RoboDK station: InvertedRobot002.rdk

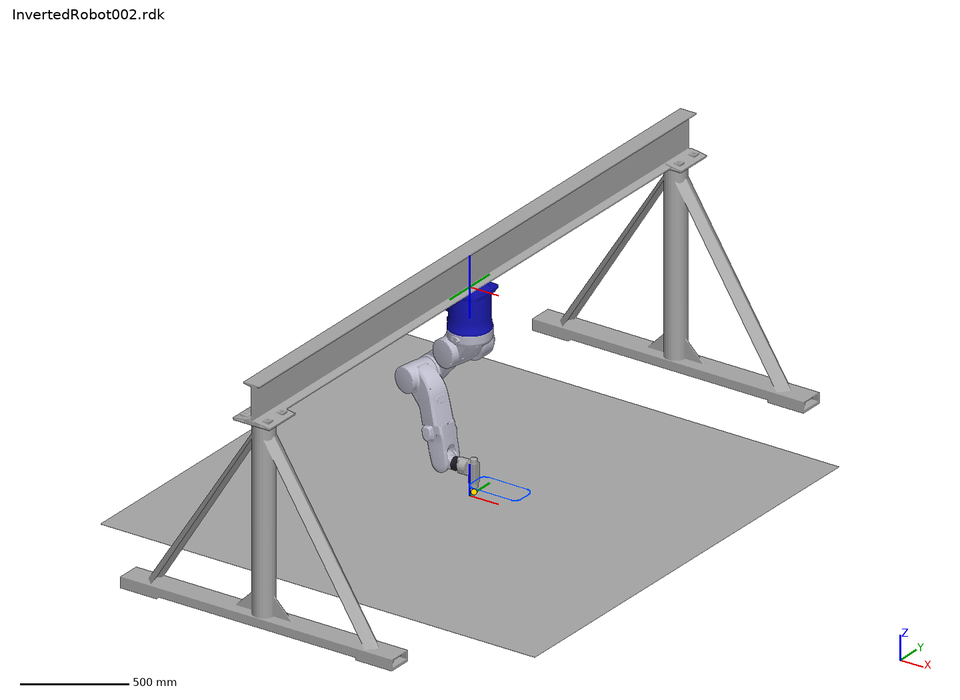
[picture v0: the station drawn from its stored meshes, robots at their saved joint values, targets as dots, program paths as lines]
Station InvertedRobot002 (saved by RoboDK 5.5.4). Poses are relative to the parent item; angles as X-Y-Z fixed-axis rotations.
Station parameters (name, value as stored): TAGS, ['Additive Manufacturing', 'Additive manufacturing'], LIN64
  - frame Denso 1 at (0, 0, 1066.8) mm, rotated rx -180 ry 0 rz 0 deg
    - robot Denso VS-6577G-B: 6 axes, payload 7 kg, reach 854 mm, repeatability 0.03 mm, weight 36 kg
        modified DH rows (alpha deg, a mm, theta deg, d mm): 0, 0, 0, 335; -90, 75, -90, 0; 0, 365, -90, 0; -90, 90, 0, 405; 90, 0, 0, 0; -90, 0, 0, 80
        joint limits [-170, -100, -119, -190, -120, -360] to [170, 135, 169, 190, 120, 360]; home [0, 0, 90, 0, 0, 0]; saved at [-167.935, 49.291, -63.192, 167.582, 76.412, 2.961]
      - tool nozzle, TCP at (110, 0, 80) mm, rotated rx 0 ry 90 rz 0 deg, size 158.8 x 76.2 x 114.9 mm, geometry from nozzle.STEP
      - tool nozzle002, TCP at (100, 0, 80) mm, rotated rx 0 ry 90 rz 0 deg, size 152.4 x 76.2 x 110.1 mm, geometry from nozzle002.STEP
  - frame Ref001 at (0, 0, 0) mm
    - object Part at (0, 0, 0) mm, size 120 x 120 x 160 mm, geometry from part.sld
  - machining project Print3D settings: /home/iRETI/RoboticsResearch/WallSections/12x12x0.875.gcode | rotZ(0) | rotX(0)*rotY(0) | rotZ(0) | on%PROGNAME%_Start | Extruder(-1) | on%PROGNAME%_Approach | on%PROGNAME%_Activate | on%PROGNAME%_Retract | on%PROGNAME%_Finish | SetRPM(%1) | SetTool(%1) | Extruder(%1) | OutOn(%1) | OutOff(%1) | OutOnMov(%1) | OutOffMov(%1) | Extruder(-1) | M_RunCode(%1)
  - program Print3D (292 instructions, listed below)
  - Python program Extruder (listed below)
  - Python program SimulateFinalResult (listed below)
  - frame Frame 4 at (0, 0, 1066.8) mm
    - object GantryAssembly at (0, 0, 0) mm, size 1524 x 3505.2 x 1270 mm, geometry from GantryAssembly.STEP
  - frame Frame 5 at (0, 0, 0) mm
    - object GarageFloor at (0, 0, 0) mm, size 2438.4 x 2438.4 x 2.5 mm, geometry from GarageFloor.STEP
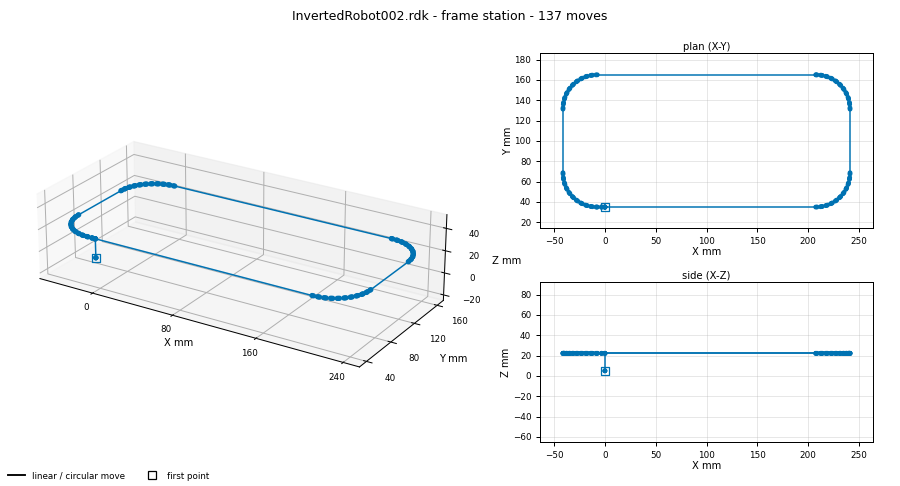
[picture p0: tool path of InvertedRobot002.rdk in frame station, 137 of 137 moves have a stored position in this frame; points joined in program order, loops and branches not executed]

--- program Print3D (robot Denso VS-6577G-B) ---
  Smooth(1)
  Call M_RunCode(107)
  Call M_RunCode(104)
  Set speed (83.3 mm/s)
  Set speed (1000.0 mm/s)
  Set Ref.: Ref001
  Set Tool: nozzle002
  Show nozzle002
  MoveJ 1 to (0, 34.91, 5) mm, rotated rx 180 ry 0 rz 180 deg; joints [-167.691, 46.522, -59.109, 167.397, 77.707, 2.725]
  MoveL 2 to (0, 34.91, 5) mm, rotated rx 180 ry 0 rz 180 deg; joints [-167.691, 46.522, -59.109, 167.397, 77.707, 2.725]
  Call Extruder(-1)
  MoveL 3 to (0, 34.91, 5) mm, rotated rx 180 ry 0 rz 180 deg; joints [-167.691, 46.522, -59.109, 167.397, 77.707, 2.725]
  Call M_RunCode(109)
  Call M_RunCode(82)
  Call Extruder(0.00000)
  Set speed (130.0 mm/s)
  MoveL 4 to (0, 34.91, 22.22) mm, rotated rx -180 ry 0 rz 180 deg; joints [-167.691, 49.055, -63.307, 167.313, 76.082, 3.099]
  Call Extruder(-2.00000)
  Set speed (40.0 mm/s)
  MoveL 5 to (0, 34.91, 22.22) mm, rotated rx -180 ry 0 rz 180 deg; joints [-167.691, 49.055, -63.307, 167.313, 76.082, 3.099]
  Call Extruder(0.00000)
  Set speed (130.0 mm/s)
  MoveL 6 to (0, 34.91, 22.22) mm, rotated rx -180 ry 0 rz 180 deg; joints [-167.691, 49.055, -63.307, 167.313, 76.082, 3.099]
  Call Extruder(2.00000)
  Set speed (40.0 mm/s)
  MoveL 7 to (0, 34.91, 22.22) mm, rotated rx -180 ry 0 rz 180 deg; joints [-167.691, 49.055, -63.307, 167.313, 76.082, 3.099]
  Set speed (30.0 mm/s)
  MoveL 8 to (0, 34.91, 22.22) mm, rotated rx -180 ry 0 rz 180 deg; joints [-167.691, 49.055, -63.307, 167.313, 76.082, 3.099]
  Call Extruder(209.10557)
  MoveL 9 to (207.51, 34.91, 22.23) mm, rotated rx -180 ry 0 rz 180 deg; joints [-36.308, 40.081, -64.789, 38.967, 109.685, 15.241]
  Call Extruder(210.41057)
  MoveL 10 to (208.82, 34.98, 22.22) mm, rotated rx 180 ry 0 rz -180 deg; joints [-35.623, 40.188, -64.796, 38.243, 109.785, 14.937]
  Call Extruder(213.89122)
  MoveL 11 to (212.3, 35.25, 22.22) mm, rotated rx -180 ry 0 rz 180 deg; joints [-33.986, 40.479, -64.812, 36.496, 109.977, 14.186]
  Call Extruder(214.76022)
  MoveL 12 to (213.16, 35.34, 22.22) mm, rotated rx -180 ry 0 rz 180 deg; joints [-33.614, 40.553, -64.815, 36.098, 110.011, 14.01]
  Call Extruder(215.62924)
  MoveL 13 to (214.01, 35.53, 22.22) mm, rotated rx -180 ry 0 rz 180 deg; joints [-33.334, 40.631, -64.819, 35.793, 110.018, 13.864]
  Call Extruder(219.10988)
  MoveL 14 to (217.4, 36.34, 22.22) mm, rotated rx 180 ry 0 rz -180 deg; joints [-32.337, 40.947, -64.83, 34.697, 110.004, 13.325]
  Call Extruder(219.97888)
  MoveL 15 to (218.25, 36.56, 22.23) mm, rotated rx -180 ry 0 rz 180 deg; joints [-32.115, 41.026, -64.832, 34.452, 109.991, 13.2]
  Call Extruder(220.84782)
  MoveL 16 to (219.06, 36.88, 22.23) mm, rotated rx -180 ry 0 rz 180 deg; joints [-31.983, 41.107, -64.834, 34.298, 109.956, 13.105]
  Call Extruder(224.32848)
  MoveL 17 to (222.28, 38.21, 22.22) mm, rotated rx -180 ry 0 rz 180 deg; joints [-31.532, 41.434, -64.839, 33.766, 109.79, 12.755]
  Call Extruder(225.19749)
  MoveL 18 to (223.08, 38.56, 22.22) mm, rotated rx 180 ry 0 rz 180 deg; joints [-31.439, 41.515, -64.839, 33.653, 109.743, 12.674]
  Call Extruder(226.06647)
  MoveL 19 to (223.83, 39, 22.22) mm, rotated rx 180 ry 0 rz -180 deg; joints [-31.427, 41.597, -64.839, 33.625, 109.678, 12.622]
  Call Extruder(229.54713)
  MoveL 20 to (226.8, 40.82, 22.22) mm, rotated rx 180 ry 0 rz 180 deg; joints [-31.43, 41.924, -64.837, 33.563, 109.403, 12.43]
  Call Extruder(230.41613)
  MoveL 21 to (227.53, 41.29, 22.23) mm, rotated rx -180 ry 0 rz 180 deg; joints [-31.443, 42.005, -64.836, 33.561, 109.332, 12.386]
  Call Extruder(231.28508)
  MoveL 22 to (228.21, 41.85, 22.23) mm, rotated rx -180 ry 0 rz 180 deg; joints [-31.529, 42.085, -64.834, 33.634, 109.245, 12.368]
  Call Extruder(234.76575)
  MoveL 23 to (230.86, 44.11, 22.22) mm, rotated rx 180 ry 0 rz 180 deg; joints [-31.903, 42.404, -64.825, 33.957, 108.893, 12.301]
  Call Extruder(235.63479)
  MoveL 24 to (231.51, 44.69, 22.23) mm, rotated rx -180 ry 0 rz 180 deg; joints [-32.002, 42.483, -64.822, 34.044, 108.804, 12.286]
  Call Extruder(236.50375)
  MoveL 25 to (232.09, 45.34, 22.22) mm, rotated rx -180 ry 0 rz 180 deg; joints [-32.168, 42.56, -64.819, 34.2, 108.703, 12.293]
  Call Extruder(239.98454)
  MoveL 26 to (234.35, 47.99, 22.23) mm, rotated rx 180 ry 0 rz 180 deg; joints [-32.84, 42.865, -64.804, 34.832, 108.295, 12.322]
  Call Extruder(240.85339)
  MoveL 27 to (234.91, 48.67, 22.22) mm, rotated rx -180 ry 0 rz 180 deg; joints [-33.011, 42.94, -64.8, 34.992, 108.193, 12.329]
  Call Extruder(241.72239)
  MoveL 28 to (235.38, 49.4, 22.23) mm, rotated rx -180 ry 0 rz 180 deg; joints [-33.239, 43.012, -64.795, 35.212, 108.082, 12.355]
  Call Extruder(245.20303)
  MoveL 29 to (237.2, 52.37, 22.22) mm, rotated rx 180 ry 0 rz 180 deg; joints [-34.153, 43.298, -64.774, 36.093, 107.636, 12.455]
  Call Extruder(246.07200)
  MoveL 30 to (237.64, 53.12, 22.22) mm, rotated rx -180 ry 0 rz 180 deg; joints [-34.381, 43.369, -64.769, 36.312, 107.526, 12.478]
  Call Extruder(246.94105)
  MoveL 31 to (237.99, 53.92, 22.23) mm, rotated rx 180 ry 0 rz 180 deg; joints [-34.66, 43.435, -64.763, 36.584, 107.407, 12.519]
  Call Extruder(250.42170)
  MoveL 32 to (239.32, 57.14, 22.23) mm, rotated rx -180 ry 0 rz 180 deg; joints [-35.769, 43.699, -64.739, 37.663, 106.936, 12.672]
  Call Extruder(251.29060)
  MoveL 33 to (239.64, 57.95, 22.22) mm, rotated rx -180 ry 0 rz 180 deg; joints [-36.043, 43.764, -64.732, 37.929, 106.819, 12.707]
  Call Extruder(252.15951)
  MoveL 34 to (239.86, 58.8, 22.23) mm, rotated rx -180 ry 0 rz -180 deg; joints [-36.362, 43.824, -64.726, 38.242, 106.697, 12.758]
  Call Extruder(255.64017)
  MoveL 35 to (240.67, 62.19, 22.22) mm, rotated rx 180 ry 0 rz -180 deg; joints [-37.627, 44.061, -64.699, 39.479, 106.21, 12.95]
  Call Extruder(256.50930)
  MoveL 36 to (240.86, 63.04, 22.22) mm, rotated rx 180 ry 0 rz 180 deg; joints [-37.94, 44.12, -64.692, 39.784, 106.089, 12.994]
  Call Extruder(257.37833)
  MoveL 37 to (240.94, 63.9, 22.22) mm, rotated rx 180 ry 0 rz -180 deg; joints [-38.29, 44.173, -64.686, 40.128, 105.964, 13.052]
  Call Extruder(260.85898)
  MoveL 38 to (241.22, 67.38, 22.22) mm, rotated rx 180 ry 0 rz 180 deg; joints [-39.68, 44.383, -64.659, 41.49, 105.468, 13.272]
  Call Extruder(262.16396)
  MoveL 39 to (241.29, 68.69, 22.22) mm, rotated rx -180 ry 0 rz 180 deg; joints [-40.198, 44.461, -64.648, 41.997, 105.283, 13.35]
  Call Extruder(324.66760)
  MoveL 40 to (241.29, 131.31, 22.23) mm, rotated rx 180 ry 0 rz 180 deg; joints [-58.241, 48.363, -63.613, 59.153, 97.958, 13.051]
  Call Extruder(325.97258)
  MoveL 41 to (241.22, 132.62, 22.22) mm, rotated rx 180 ry 0 rz 180 deg; joints [-58.516, 48.444, -63.579, 59.409, 97.837, 12.988]
  Call Extruder(329.45322)
  MoveL 42 to (240.94, 136.1, 22.22) mm, rotated rx -180 ry 0 rz -180 deg; joints [-59.257, 48.656, -63.489, 60.103, 97.519, 12.822]
  Call Extruder(330.32226)
  MoveL 43 to (240.86, 136.96, 22.22) mm, rotated rx -180 ry 0 rz 180 deg; joints [-59.443, 48.708, -63.466, 60.278, 97.441, 12.78]
  Call Extruder(331.19137)
  MoveL 44 to (240.67, 137.81, 22.22) mm, rotated rx 180 ry 0 rz 180 deg; joints [-59.656, 48.756, -63.445, 60.479, 97.36, 12.748]
  Call Extruder(334.67203)
  MoveL 45 to (239.86, 141.2, 22.22) mm, rotated rx 180 ry 0 rz 180 deg; joints [-60.509, 48.942, -63.36, 61.288, 97.041, 12.614]
  Call Extruder(335.54095)
  MoveL 46 to (239.64, 142.05, 22.22) mm, rotated rx -180 ry 0 rz -180 deg; joints [-60.723, 48.988, -63.339, 61.491, 96.962, 12.58]
  Call Extruder(336.40987)
  MoveL 47 to (239.32, 142.86, 22.22) mm, rotated rx -180 ry 0 rz -180 deg; joints [-60.959, 49.029, -63.32, 61.717, 96.882, 12.555]
  Call Extruder(339.89051)
  MoveL 48 to (237.99, 146.08, 22.22) mm, rotated rx -180 ry 0 rz 180 deg; joints [-61.903, 49.188, -63.243, 62.621, 96.567, 12.453]
  Call Extruder(340.75954)
  MoveL 49 to (237.64, 146.88, 22.22) mm, rotated rx -180 ry 0 rz 180 deg; joints [-62.139, 49.227, -63.224, 62.846, 96.49, 12.428]
  Call Extruder(341.62850)
  MoveL 50 to (237.2, 147.63, 22.22) mm, rotated rx -180 ry 0 rz 180 deg; joints [-62.394, 49.261, -63.207, 63.092, 96.413, 12.411]
  Call Extruder(345.10915)
  MoveL 51 to (235.38, 150.6, 22.22) mm, rotated rx -180 ry 0 rz -180 deg; joints [-63.412, 49.391, -63.142, 64.073, 96.107, 12.343]
  Call Extruder(345.97817)
  MoveL 52 to (234.91, 151.33, 22.22) mm, rotated rx -180 ry 0 rz 180 deg; joints [-63.666, 49.423, -63.125, 64.318, 96.032, 12.326]
  Call Extruder(346.84712)
  MoveL 53 to (234.35, 152.01, 22.22) mm, rotated rx 180 ry 0 rz 180 deg; joints [-63.935, 49.449, -63.112, 64.578, 95.957, 12.318]
  Call Extruder(350.32775)
  MoveL 54 to (232.09, 154.66, 22.22) mm, rotated rx 180 ry 0 rz 180 deg; joints [-65.009, 49.55, -63.06, 65.619, 95.664, 12.285]
  Call Extruder(351.19679)
  MoveL 55 to (231.51, 155.31, 22.22) mm, rotated rx 180 ry 0 rz -180 deg; joints [-65.277, 49.575, -63.047, 65.879, 95.591, 12.276]
  Call Extruder(352.06577)
  MoveL 56 to (230.86, 155.89, 22.22) mm, rotated rx 180 ry 0 rz -180 deg; joints [-65.556, 49.593, -63.037, 66.15, 95.521, 12.277]
  Call Extruder(355.54644)
  MoveL 57 to (228.21, 158.15, 22.22) mm, rotated rx -180 ry 0 rz 180 deg; joints [-66.671, 49.664, -62.999, 67.235, 95.241, 12.28]
  Call Extruder(356.41541)
  MoveL 58 to (227.54, 158.71, 22.22) mm, rotated rx 180 ry 0 rz -180 deg; joints [-66.949, 49.681, -62.99, 67.505, 95.172, 12.28]
  Call Extruder(357.28446)
  MoveL 59 to (226.8, 159.18, 22.22) mm, rotated rx -180 ry 0 rz 180 deg; joints [-67.233, 49.691, -62.985, 67.783, 95.105, 12.29]
  Call Extruder(360.76512)
  MoveL 60 to (223.83, 161, 22.23) mm, rotated rx -180 ry 0 rz 180 deg; joints [-68.374, 49.731, -62.963, 68.897, 94.839, 12.33]
  Call Extruder(361.63406)
  MoveL 61 to (223.08, 161.44, 22.22) mm, rotated rx -180 ry 0 rz 180 deg; joints [-68.659, 49.741, -62.958, 69.175, 94.773, 12.34]
  Call Extruder(362.50303)
  MoveL 62 to (222.28, 161.79, 22.22) mm, rotated rx 180 ry 0 rz -180 deg; joints [-68.946, 49.743, -62.956, 69.456, 94.71, 12.359]
  Call Extruder(365.98369)
  MoveL 63 to (219.06, 163.12, 22.22) mm, rotated rx 180 ry 0 rz -180 deg; joints [-70.098, 49.752, -62.952, 70.584, 94.458, 12.437]
  Call Extruder(366.85268)
  MoveL 64 to (218.25, 163.44, 22.22) mm, rotated rx -180 ry 0 rz -180 deg; joints [-70.385, 49.754, -62.951, 70.865, 94.396, 12.456]
  Call Extruder(367.72170)
  MoveL 65 to (217.4, 163.66, 22.23) mm, rotated rx -180 ry 0 rz -180 deg; joints [-70.671, 49.748, -62.954, 71.146, 94.336, 12.485]
  Call Extruder(371.20234)
  MoveL 66 to (214.01, 164.47, 22.22) mm, rotated rx -180 ry 0 rz 180 deg; joints [-71.82, 49.726, -62.966, 72.273, 94.098, 12.601]
  Call Extruder(372.07132)
  MoveL 67 to (213.16, 164.66, 22.22) mm, rotated rx -180 ry 0 rz 180 deg; joints [-72.107, 49.72, -62.969, 72.554, 94.038, 12.63]
  Call Extruder(372.94029)
  MoveL 68 to (212.3, 164.75, 22.22) mm, rotated rx 180 ry 0 rz -180 deg; joints [-72.389, 49.707, -62.976, 72.831, 93.982, 12.668]
  Call Extruder(376.42094)
  MoveL 69 to (208.82, 165.02, 22.22) mm, rotated rx 180 ry 0 rz -180 deg; joints [-73.52, 49.653, -63.005, 73.942, 93.756, 12.822]
  Call Extruder(377.28995)
  MoveL 70 to (207.95, 165.07, 22.22) mm, rotated rx 180 ry 0 rz -180 deg; joints [-73.802, 49.639, -63.012, 74.219, 93.699, 12.86]
  Call Extruder(377.72605)
  MoveL 71 to (207.51, 165.09, 22.23) mm, rotated rx 180 ry 0 rz 180 deg; joints [-73.944, 49.632, -63.016, 74.358, 93.671, 12.88]
  Call Extruder(592.33024)
  MoveL 72 to (-7.51, 165.09, 22.22) mm, rotated rx -180 ry 0 rz -180 deg; joints [-135.418, 53.569, -59.808, 135.248, 85.561, 4.388]
  Call Extruder(593.63529)
  MoveL 73 to (-8.82, 165.02, 22.22) mm, rotated rx -180 ry 0 rz 180 deg; joints [-135.652, 53.616, -59.752, 135.488, 85.616, 4.297]
  Call Extruder(597.11593)
  MoveL 74 to (-12.3, 164.75, 22.22) mm, rotated rx 180 ry 0 rz -180 deg; joints [-136.283, 53.737, -59.603, 136.133, 85.764, 4.061]
  Call Extruder(597.98490)
  MoveL 75 to (-13.16, 164.66, 22.22) mm, rotated rx -180 ry 0 rz 180 deg; joints [-136.442, 53.767, -59.566, 136.295, 85.801, 4.004]
  Call Extruder(598.85386)
  MoveL 76 to (-14.01, 164.47, 22.22) mm, rotated rx 180 ry 0 rz 180 deg; joints [-136.614, 53.792, -59.534, 136.47, 85.83, 3.951]
  Call Extruder(602.33452)
  MoveL 77 to (-17.4, 163.66, 22.22) mm, rotated rx 180 ry 0 rz 180 deg; joints [-137.308, 53.891, -59.408, 137.175, 85.948, 3.747]
  Call Extruder(603.20352)
  MoveL 78 to (-18.25, 163.44, 22.22) mm, rotated rx 180 ry 0 rz -180 deg; joints [-137.481, 53.915, -59.376, 137.351, 85.977, 3.697]
  Call Extruder(604.07254)
  MoveL 79 to (-19.06, 163.12, 22.22) mm, rotated rx 180 ry 0 rz -180 deg; joints [-137.666, 53.935, -59.351, 137.539, 85.999, 3.654]
  Call Extruder(607.55321)
  MoveL 80 to (-22.28, 161.79, 22.22) mm, rotated rx -180 ry 0 rz 180 deg; joints [-138.408, 54.011, -59.25, 138.289, 86.084, 3.484]
  Call Extruder(608.42217)
  MoveL 81 to (-23.08, 161.44, 22.23) mm, rotated rx -180 ry 0 rz 180 deg; joints [-138.594, 54.029, -59.226, 138.477, 86.105, 3.442]
  Call Extruder(609.29114)
  MoveL 82 to (-23.83, 161, 22.22) mm, rotated rx -180 ry 0 rz -180 deg; joints [-138.788, 54.043, -59.207, 138.672, 86.117, 3.408]
  Call Extruder(612.77178)
  MoveL 83 to (-26.8, 159.18, 22.23) mm, rotated rx 180 ry 0 rz 180 deg; joints [-139.565, 54.096, -59.136, 139.456, 86.166, 3.273]
  Call Extruder(613.64080)
  MoveL 84 to (-27.54, 158.71, 22.22) mm, rotated rx -180 ry 0 rz 180 deg; joints [-139.759, 54.109, -59.118, 139.651, 86.178, 3.241]
  Call Extruder(614.50982)
  MoveL 85 to (-28.21, 158.15, 22.22) mm, rotated rx -180 ry 0 rz 180 deg; joints [-139.959, 54.117, -59.107, 139.852, 86.181, 3.216]
  Call Extruder(617.99048)
  MoveL 86 to (-30.86, 155.89, 22.22) mm, rotated rx -180 ry 0 rz 180 deg; joints [-140.759, 54.146, -59.067, 140.655, 86.191, 3.117]
  Call Extruder(618.85941)
  MoveL 87 to (-31.51, 155.31, 22.23) mm, rotated rx -180 ry 0 rz 180 deg; joints [-140.959, 54.153, -59.057, 140.856, 86.193, 3.093]
  Call Extruder(619.72839)
  MoveL 88 to (-32.09, 154.66, 22.22) mm, rotated rx 180 ry 0 rz -180 deg; joints [-141.161, 54.155, -59.054, 141.058, 86.186, 3.077]
  Call Extruder(623.20904)
  MoveL 89 to (-34.35, 152.01, 22.22) mm, rotated rx 180 ry 0 rz 180 deg; joints [-141.97, 54.161, -59.046, 141.869, 86.154, 3.014]
  Call Extruder(624.07805)
  MoveL 90 to (-34.91, 151.34, 22.23) mm, rotated rx 180 ry 0 rz -180 deg; joints [-142.173, 54.163, -59.044, 142.072, 86.146, 2.998]
  Call Extruder(624.94703)
  MoveL 91 to (-35.38, 150.6, 22.22) mm, rotated rx -180 ry 0 rz -180 deg; joints [-142.374, 54.159, -59.05, 142.273, 86.128, 2.99]
  Call Extruder(628.42769)
  MoveL 92 to (-37.2, 147.63, 22.22) mm, rotated rx -180 ry 0 rz -180 deg; joints [-143.18, 54.141, -59.073, 143.078, 86.054, 2.96]
  Call Extruder(629.29668)
  MoveL 93 to (-37.64, 146.88, 22.22) mm, rotated rx -180 ry 0 rz -180 deg; joints [-143.382, 54.137, -59.08, 143.28, 86.034, 2.953]
  Call Extruder(630.16566)
  MoveL 94 to (-37.99, 146.08, 22.22) mm, rotated rx -180 ry 0 rz 180 deg; joints [-143.579, 54.127, -59.093, 143.476, 86.006, 2.953]
  Call Extruder(633.64631)
  MoveL 95 to (-39.32, 142.86, 22.22) mm, rotated rx 180 ry 0 rz 180 deg; joints [-144.37, 54.086, -59.149, 144.264, 85.887, 2.954]
  Call Extruder(634.51530)
  MoveL 96 to (-39.64, 142.05, 22.22) mm, rotated rx -180 ry 0 rz 180 deg; joints [-144.568, 54.076, -59.163, 144.461, 85.857, 2.954]
  Call Extruder(635.38427)
  MoveL 97 to (-39.86, 141.2, 22.22) mm, rotated rx 180 ry 0 rz -180 deg; joints [-144.758, 54.06, -59.184, 144.65, 85.817, 2.962]
  Call Extruder(638.86493)
  MoveL 98 to (-40.67, 137.81, 22.22) mm, rotated rx 180 ry 0 rz -180 deg; joints [-145.521, 53.996, -59.269, 145.407, 85.655, 2.991]
  Call Extruder(639.73393)
  MoveL 99 to (-40.86, 136.96, 22.22) mm, rotated rx -180 ry 0 rz 180 deg; joints [-145.711, 53.98, -59.291, 145.596, 85.614, 2.998]
  Call Extruder(640.60294)
  MoveL 100 to (-40.95, 136.1, 22.22) mm, rotated rx -180 ry 0 rz -180 deg; joints [-145.891, 53.959, -59.319, 145.774, 85.564, 3.012]
  Call Extruder(644.08358)
  MoveL 101 to (-41.22, 132.62, 22.23) mm, rotated rx -180 ry 0 rz -180 deg; joints [-146.612, 53.872, -59.432, 146.488, 85.359, 3.067]
  Call Extruder(645.38859)
  MoveL 102 to (-41.29, 131.31, 22.22) mm, rotated rx -180 ry 0 rz 180 deg; joints [-146.881, 53.838, -59.476, 146.754, 85.281, 3.087]
  Call Extruder(707.89230)
  MoveL 103 to (-41.29, 68.69, 22.22) mm, rotated rx 180 ry 0 rz 180 deg; joints [-161.158, 52.302, -61.135, 160.949, 81.644, 2.873]
  Call Extruder(709.19730)
  MoveL 104 to (-41.22, 67.38, 22.22) mm, rotated rx 180 ry 0 rz -180 deg; joints [-161.486, 52.273, -61.161, 161.277, 81.576, 2.843]
  Call Extruder(712.67795)
  MoveL 105 to (-40.95, 63.9, 22.22) mm, rotated rx -180 ry 0 rz 180 deg; joints [-162.358, 52.193, -61.233, 162.151, 81.388, 2.761]
  Call Extruder(713.54695)
  MoveL 106 to (-40.86, 63.04, 22.22) mm, rotated rx -180 ry 0 rz -180 deg; joints [-162.576, 52.172, -61.251, 162.369, 81.341, 2.739]
  Call Extruder(714.41596)
  MoveL 107 to (-40.67, 62.19, 22.22) mm, rotated rx -180 ry 0 rz 180 deg; joints [-162.782, 52.146, -61.274, 162.575, 81.285, 2.723]
  Call Extruder(717.89661)
  MoveL 108 to (-39.86, 58.8, 22.22) mm, rotated rx -180 ry 0 rz 180 deg; joints [-163.607, 52.04, -61.367, 163.399, 81.055, 2.654]
  Call Extruder(718.76559)
  MoveL 109 to (-39.64, 57.95, 22.22) mm, rotated rx -180 ry 0 rz -180 deg; joints [-163.813, 52.013, -61.391, 163.605, 80.997, 2.636]
  Call Extruder(719.63456)
  MoveL 110 to (-39.32, 57.14, 22.22) mm, rotated rx -180 ry 0 rz 180 deg; joints [-164.003, 51.98, -61.418, 163.795, 80.93, 2.623]
  Call Extruder(723.11522)
  MoveL 111 to (-37.99, 53.92, 22.23) mm, rotated rx -180 ry 0 rz -180 deg; joints [-164.765, 51.848, -61.53, 164.556, 80.662, 2.567]
  Call Extruder(723.98421)
  MoveL 112 to (-37.64, 53.12, 22.22) mm, rotated rx -180 ry 0 rz 180 deg; joints [-164.955, 51.814, -61.557, 164.745, 80.594, 2.552]
  Call Extruder(724.85321)
  MoveL 113 to (-37.2, 52.37, 22.23) mm, rotated rx -180 ry 0 rz -180 deg; joints [-165.127, 51.776, -61.589, 164.916, 80.519, 2.542]
  Call Extruder(728.33386)
  MoveL 114 to (-35.38, 49.4, 22.22) mm, rotated rx 180 ry 0 rz 180 deg; joints [-165.811, 51.619, -61.715, 165.597, 80.215, 2.499]
  Call Extruder(729.20284)
  MoveL 115 to (-34.91, 48.66, 22.22) mm, rotated rx -180 ry 0 rz -180 deg; joints [-165.981, 51.58, -61.747, 165.766, 80.139, 2.488]
  Call Extruder(730.07182)
  MoveL 116 to (-34.35, 47.99, 22.22) mm, rotated rx -180 ry 0 rz -180 deg; joints [-166.129, 51.535, -61.781, 165.914, 80.056, 2.481]
  Call Extruder(733.55248)
  MoveL 117 to (-32.09, 45.34, 22.22) mm, rotated rx -180 ry 0 rz 180 deg; joints [-166.719, 51.356, -61.918, 166.499, 79.723, 2.453]
  Call Extruder(734.42146)
  MoveL 118 to (-31.51, 44.69, 22.22) mm, rotated rx -180 ry 0 rz -180 deg; joints [-166.865, 51.311, -61.952, 166.643, 79.64, 2.445]
  Call Extruder(735.29045)
  MoveL 119 to (-30.86, 44.11, 22.22) mm, rotated rx -180 ry 0 rz -180 deg; joints [-166.986, 51.261, -61.989, 166.763, 79.551, 2.443]
  Call Extruder(738.77110)
  MoveL 120 to (-28.21, 41.85, 22.23) mm, rotated rx -180 ry 0 rz 180 deg; joints [-167.465, 51.062, -62.133, 167.235, 79.195, 2.432]
  Call Extruder(739.64010)
  MoveL 121 to (-27.53, 41.29, 22.22) mm, rotated rx -180 ry 0 rz -180 deg; joints [-167.582, 51.011, -62.169, 167.351, 79.106, 2.429]
  Call Extruder(740.50907)
  MoveL 122 to (-26.8, 40.82, 22.22) mm, rotated rx -180 ry 0 rz -180 deg; joints [-167.672, 50.957, -62.207, 167.438, 79.013, 2.432]
  Call Extruder(743.98973)
  MoveL 123 to (-23.83, 39, 22.22) mm, rotated rx -180 ry 0 rz 180 deg; joints [-168.021, 50.74, -62.354, 167.778, 78.642, 2.443]
  Call Extruder(744.85872)
  MoveL 124 to (-23.08, 38.56, 22.22) mm, rotated rx -180 ry 0 rz -180 deg; joints [-168.106, 50.685, -62.391, 167.861, 78.549, 2.445]
  Call Extruder(745.72772)
  MoveL 125 to (-22.28, 38.21, 22.22) mm, rotated rx -180 ry 0 rz -180 deg; joints [-168.16, 50.628, -62.428, 167.912, 78.454, 2.454]
  Call Extruder(749.20838)
  MoveL 126 to (-19.06, 36.88, 22.22) mm, rotated rx -180 ry 0 rz 180 deg; joints [-168.362, 50.397, -62.575, 168.102, 78.076, 2.493]
  Call Extruder(750.07736)
  MoveL 127 to (-18.25, 36.56, 22.22) mm, rotated rx 180 ry 0 rz -180 deg; joints [-168.409, 50.339, -62.611, 168.145, 77.982, 2.503]
  Call Extruder(750.94633)
  MoveL 128 to (-17.4, 36.34, 22.22) mm, rotated rx -180 ry 0 rz 180 deg; joints [-168.423, 50.279, -62.647, 168.156, 77.887, 2.52]
  Call Extruder(754.42699)
  MoveL 129 to (-14.01, 35.53, 22.22) mm, rotated rx 180 ry 0 rz -180 deg; joints [-168.461, 50.039, -62.79, 168.178, 77.512, 2.592]
  Call Extruder(755.29600)
  MoveL 130 to (-13.16, 35.34, 22.22) mm, rotated rx -180 ry 0 rz -180 deg; joints [-168.465, 49.979, -62.825, 168.177, 77.418, 2.611]
  Call Extruder(756.16500)
  MoveL 131 to (-12.3, 35.25, 22.22) mm, rotated rx -180 ry 0 rz -180 deg; joints [-168.436, 49.919, -62.859, 168.143, 77.327, 2.637]
  Call Extruder(759.64564)
  MoveL 132 to (-8.82, 34.98, 22.23) mm, rotated rx 180 ry 0 rz 180 deg; joints [-168.293, 49.676, -62.993, 167.979, 76.965, 2.75]
  Call Extruder(760.51461)
  MoveL 133 to (-7.95, 34.93, 22.23) mm, rotated rx -180 ry 0 rz 180 deg; joints [-168.251, 49.615, -63.026, 167.931, 76.875, 2.78]
  Call Extruder(760.95070)
  MoveL 134 to (-7.51, 34.91, 22.23) mm, rotated rx 180 ry 0 rz 180 deg; joints [-168.227, 49.584, -63.042, 167.905, 76.831, 2.795]
  Call Extruder(765.12213)
  MoveL 135 to (-3.33, 34.91, 22.22) mm, rotated rx 180 ry 0 rz -180 deg; joints [-167.935, 49.291, -63.192, 167.582, 76.412, 2.961]
  Call Extruder(763.12213)
  Set speed (40.0 mm/s)
  MoveL 136 to (-3.33, 34.91, 22.22) mm, rotated rx 180 ry 0 rz -180 deg; joints [-167.935, 49.291, -63.192, 167.582, 76.412, 2.961]
  Set speed (1000.0 mm/s)
  Call Extruder(-1)
  MoveL 137 to (-3.33, 34.91, 22.22) mm, rotated rx 180 ry 0 rz -180 deg; joints [-167.935, 49.291, -63.192, 167.582, 76.412, 2.961]
  Call Extruder(0.00000)
  Call M_RunCode(104)
  Call M_RunCode(84)
  Call M_RunCode(140)

--- Python program Extruder ---
# This macro allows simulating a 3D printing extruder
# The macro will output spray gun statistics
#
# More information about the RoboDK API here:
# https://robodk.com/doc/en/RoboDK-API.html
# For more information visit:
# http://www.robodk.com/doc/en/PythonAPI/robolink.html
#
# Define the default action (0 to deactivate, +1 to activate, -1 to clear any spray gun simulation)
# Setting it to None will display a message
ACTION = None
# Check if we are running this program inside another program and passing arguments
import sys
if len(sys.argv) > 1:
    ACTION = float(sys.argv[1])
    # For faster speed: igone values greater than 0
    if ACTION > 0:
        quit()

from robolink import *    # API to communicate with RoboDK
from robodk import *      # basic matrix operations
RDK = Robolink()

# quit if we are not in simulation mode
if RDK.RunMode() != RUNMODE_SIMULATE:
    quit()

# Get any previously added spray gun simulations and display statistics (spray on the part vs spray falling out of the part)
existing_material_simulation = False
info, stats_data = RDK.Spray_GetStats()
if stats_data.size(1) > 0:
    print("Spray gun statistics:")
    print(info)
    print(stats_data.tr())
    existing_material_simulation = True
    # # Diplay statistics
    # RDK.ShowMessage("Material used: %.1f%%<br>Material waisted: %.1f%%<br>Total particles: %.1f" % (data[1,0],data[2,0],data[3,0]), True)
    # # Clear previous spray
    # RDK.Spray_Clear()

# If the default ACTION is None, display a message to activate/deactivate the spray gun
if ACTION is None:
    print('Note: This macro can be called as Extruder(0) to turn it ON or Extruder(-1) to turn it OFF')
    entry = mbox('Turn Extruder ON or OFF', ('On', '0'), ('Off', '-1'))
    if not entry:
        quit()
    ACTION = int(entry)

if ACTION < 0:
    # Turn material deposition off
    # Select Escape to delete existing material simulations
    #RDK.Spray_Clear()
    RDK.Spray_SetState(SPRAY_OFF)

elif ACTION >= 0:

    if existing_material_simulation:
        # Select Esc key to delete existing material simulations and force a new type of spray gun simulation
        RDK.Spray_SetState(SPRAY_ON)
        exit()


    # Create a new spray gun object in RoboDK for material deposition (3D printing simulation)
    # by using RDK.Spray_Add(tool, object, options_command, volume, geometry)
    # tool: tool item (TCP) to use
    # object: object to project the particles
    # options_command (optional): string to specify options. Example:
    #     STEP=AxB: Defines the grid to be projected 1x1 means only one line of particle projection (for example, for welding)
    #     PARTICLE: Defines the shape and size of particle (sphere or particle), unless a specific geometry is provided:
    #       a- SPHERE(radius, facets)
    #       b- SPHERE(radius, facets, scalex, scaley, scalez)
    #       b- CUBE(sizex, sizey, sizez)
    #     RAND=factor: Defines a random factor factor 0 means that the particles are not deposited randomly
    #     ELLYPSE: defines the volume as an ellypse (default)
    #     RECTANGLE: defines the volume as a rectangle
    #     PROJECT: project the particles to the surface (default) (for welding, painting or scanning)
    #     NO_PROJECT: does not project the particles to the surface (for example, for 3D printing)
    #
    # volume (optional): Matrix of parameters defining the volume of the spray gun
    # geometry (optional): Matrix of vertices defining the triangles.


    diameter = 22.225 # in mm
    detail = 8 # number of rings of detail to display the sphere
    scale = '1,1,0.5' # scale the particle in 0.5 along the tool Z axis (simulating gravity effect)
    options_command = "ELLYPSE NO_PROJECT PARTICLE=SPHERE(%.3f,%.0f,%s)" % (diameter, detail, scale) # simulate
    #options_command = "PARTICLE=CUBE(10,10,2) STEP=8x8"
    #options_command = "PARTICLE=SPHERE(4,8) STEP=8x8"
    #options_command = "PARTICLE=SPHERE(4,8,1,1,0.1) STEP=8x8 RAND=3"

    # Example commands for welding:
    # options_command = "PROJECT PARTICLE=SPHERE(4,8)"
    # options_command = PARTICLE=SPHERE(4,8) STEP=1x0

    tool = 0    # auto detect active tool
    obj = 0     # auto detect object in active reference frame

    # Material is deposited at 0,0,0 with respect to the TCP coordinates
    close_param = [0,0,0,  0,0,0,  0,0,0,     0.7,0.5,0.8,1] # color as RGBA
    far_param   = [0,0,0,  0,0,0,  0,0,0,     0.7,0.5,0.8,1] # color as RGBA
    volume = Mat([close_param, far_param])
    RDK.Spray_Add(tool, obj, options_command, volume.tr())
    RDK.Spray_SetState(SPRAY_ON)

--- Python program SimulateFinalResult ---
# This script will simulate the final result of the 3D printed part using the Spray function

# Or visit: http://www.robodk.com/doc/PythonAPI/
# Note: you do not need to keep a copy of this file, your python script is saved with the station
from robolink import *    # API to communicate with RoboDK
from robodk import *      # basic matrix operations


RENDER = True      # Set to False
STEP_MM = 2         # Detail step in MM for linear moves
STEP_DEG = 2        # Detail step in DEG for joint moves

# Start a connection with the RoboDK API
RDK = Robolink()

# Select the first/only robot in the cell:
program = RDK.ItemUserPick('Select a program to simulate', ITEM_TYPE_PROGRAM)
if not program.Valid():
    raise Exception("No program available")

# Get the robot
robot = RDK.Item('', ITEM_TYPE_ROBOT)
#robot = program.getLink(ITEM_TYPE_ROBOT) # available in newer versions
if not robot.Valid():
    raise Exception("No robot available")

progname = program.Name()
print("Using program %s" % progname)


# Get the program as a list of joint values
tool = robot.getLink(ITEM_TYPE_TOOL)
progok_jlist = program.InstructionListJoints(STEP_MM, STEP_DEG)
progok = progok_jlist[0] # progok: String that indicates if there are any issues with the program
jlist = progok_jlist[1]  # jlist: list of joints

# Check that the program is correct and has at least a movement
njoints = jlist.size(1)
if njoints < 1:
    raise Exception("Program %s has no movements" % name)

# Check if there are any issues with the program:
if progok != "Success":
    raise Exception("Problems with program %s: %s." %(name, progok))

# Reset any material deposition simulation
RDK.Spray_Clear()

robot.setPoseTool(tool)

# Start material deposition simulation according to the Extruder script
RDK.RunProgram('Extruder(0)')
# Alternatively:
#RDK.Item('Extruder', ITEM_TYPE_PYTHON).RunProgram([1])

if not RENDER:
    RDK.Render(False)

# Iterate through all joints in the matrix and check for collisions
njoints_all = jlist.size(1)
for i in range(njoints_all):
    ji = jlist[:,i].tolist()

    # Update the robot to a new position (it will create a new particle)
    robot.setJoints(ji)
    if not RENDER:
        # If Render is turned off (faster) update the position to draw a new particle
        RDK.Update()

    # Show a message in the RoboDK status bar from time to time
    if i % 10 == 0:
        msg = "Quick material deposition simulation for %s (%.1f %%)" % (progname, 100.0*(i/njoints_all))
        print(msg)
        RDK.ShowMessage(msg, False)

    # Render from time to time even if we have render deactivated
    if not RENDER and i % 500 == 0:
        RDK.Render()

RDK.Render(True)
msg = "Done"
print("Done")
RDK.ShowMessage(msg, False)
